{attribute 'GeneratedUsingTerminal: EL2262-0000-0002'}
{attribute addProperty BoxType "EL2262-0000-0002"}
{attribute addProperty Id "Cycle_Counter1AT %Q*UINT2"}
{attribute addProperty CRC "2830499814"}
{attribute addProperty Size "2"}
TYPE CycCount1_A8B5FFE6 :
STRUCT
	{attribute addProperty Name "Cycle_Counter1"}
	Cycle_Counter1 AT %Q* : UINT;
END_STRUCT
END_TYPE

(* stored: Version 1.2.0.0, ProductVersion 3.1.4024.9
   DUT CycCount1_A8B5FFE6: Id {dd84592a-601c-4e2e-905d-22305a313481} *)
